FUNCTION_BLOCK FB_ButtonToggle
VAR_INPUT
	bReset  :BOOL;
	bEnable :BOOL := TRUE;
	bButt   :BOOL;
END_VAR
VAR
	fbButt  :R_TRIG;
END_VAR
VAR_OUTPUT
	bOutB   :BOOL;
END_VAR

fbButt(CLK:=bButt);

IF fbButt.Q AND bEnable THEN
	IF bOutB THEN bOutB := FALSE;
		ELSE bOutB := TRUE;
	END_IF
END_IF

IF bReset THEN bOutB := FALSE;
END_IF

END_FUNCTION_BLOCK

(* stored: Version 1.1.0.1, ProductVersion 3.1.4024.4
   POU FB_ButtonToggle: Id {cd045b62-cdd8-44e2-8806-19439e36e62d}, SpecialFunc None *)
